// TwinCAT 3 PLC project VGR0
// ProgramVersion: 3.1.4024.0
// libraries:
//   Tc2_Standard, * (Beckhoff Automation GmbH)
//   Tc2_System, * (Beckhoff Automation GmbH)
//   Tc3_Module, * (Beckhoff Automation GmbH)
// project tree:
//   DUTs/ ST_Axis.TcDUT
//   GVLs/ Axis.TcGVL (not stored) (excluded from build), INPUT.TcGVL, OUTPUT.TcGVL, Settings.TcGVL, VGR.TcGVL
//   POUs/ AxisHorizontal.TcPOU, AxisRotate.TcPOU, AxisVertical.TcPOU, MAIN_10MS.TcPOU, MAIN_1MS.TcPOU, Motor_move.TcPOU, StateMachine.TcPOU
//   POUs/FBs/ AboutEqual.TcPOU, AxisMovementController.TcPOU, AxisReferencing.TcPOU, EncoderSignalProcessor.TcPOU, Motor_Direction.TcPOU, Motor_Enable.TcPOU
//   / VGR_10MS.TcTTO, VGR_1MS.TcTTO
// (motion and I/O tree: see PLC project vgr)
// real-time tasks:
//   TASK PlcTask: cycle T#10ms, priority 20, ADS port 350
//   TASK VGR_10MS: cycle T#10ms, priority 22, ADS port 352
//   TASK VGR_1MS: cycle T#1ms, priority 23, ADS port 353
// variable links:
//   VGR0/VGR0 Instance <-> Device 1 (EtherCAT)/Term 1 (EK1100)/Term 6 (EL5152)
//     VGR_10MS Inputs/INPUT.IW_VGR_CounterValueHorizontal <-> ENC Status compact Channel 2/Counter value
//     VGR_10MS Inputs/INPUT.IW_VGR_CounterValueVertical <-> ENC Status compact Channel 1/Counter value
//   VGR0/VGR0 Instance <-> Device 1 (EtherCAT)/Term 1 (EK1100)/Term 7 (EL5152)
//     VGR_10MS Inputs/INPUT.IW_VGR_CounterValueRotate <-> ENC Status compact Channel 1/Counter value

CONFIGURATION VGR0
    RESOURCE PLC ON TwinCAT3
        TASK VGR_10MS(INTERVAL := T#10ms, PRIORITY := 22);
        TASK VGR_1MS(INTERVAL := T#1ms, PRIORITY := 23);
        PROGRAM MAIN_10MS WITH VGR_10MS : MAIN_10MS;
        PROGRAM MAIN WITH VGR_10MS : MAIN;
        PROGRAM MAIN_1MS WITH VGR_1MS : MAIN_1MS;
    END_RESOURCE
END_CONFIGURATION

// ---- DUTs/ST_Axis.TcDUT
TYPE ST_Axis :
STRUCT
	uiCounterValue				  		: UINT;
	bSetCounter				 			: BOOL;
	uiSetCounterValue			 		: UINT := 0;
	iControl 							: INT; //VGR = PWM Motor M1 vertical axis enable at 10#32
	iPWM				 				: INT; //VGR = PWM Motor M1 vertical axis
	bJogMinus					 		: BOOL; //VGR - Q1 = Motor M1 vertical axis up
	bJogPlus					 		: BOOL; //VGR - Q2 = Motor M1 vertical axis down
END_STRUCT
END_TYPE

// ---- GVLs/INPUT.TcGVL
{attribute 'qualified_only'}
VAR_GLOBAL
IX_START AT %I*: BOOL;
IX_STOP AT %I*:	BOOL;
IW_VGR_CounterValueVertical  		AT %I* : UINT;
IW_VGR_CounterValueHorizontal  		AT %I* : UINT;
IW_VGR_CounterValueRotate  			AT %I* : UINT;

END_VAR

// ---- GVLs/OUTPUT.TcGVL
{attribute 'qualified_only'}
VAR_GLOBAL

QX_VGR_SetCounterVertical 			AT %Q* : BOOL;
QX_VGR_SetCounterHorizontal 		AT %Q* : BOOL;
QX_VGR_SetCounterRotate 			AT %Q* : BOOL;

QW_VGR_SetCounterValueVertical 		AT %Q* : UINT;
QW_VGR_SetCounterValueRotate 		AT %Q* : UINT;
QW_VGR_SetCounterValueHorizontal 	AT %Q* : UINT;

END_VAR

// ---- GVLs/Settings.TcGVL
{attribute 'qualified_only'}
VAR_GLOBAL
	bUseAxisVertical : BOOL := TRUE;
	bUseAxisHorizontal : BOOL := TRUE;
	bUseAxisRotate : BOOL := TRUE;
	
	CurrentState : STRING ;

	desiredSpeedVertical : INT := 5000;
	desiredSpeedHorizontal : INT := 5000;
	desiredSpeedRotation : INT := 5000;
	
	pickPositionVertical : UINT := 500;
	pickPositionHorizontal : UINT := 500;
	pickPositionRotation : UINT := 500;
	
	placePositionVertical : UINT := 100;
	placePositionHorizontal : UINT := 100;
	placePositionRotation : UINT := 200;
END_VAR

// ---- GVLs/VGR.TcGVL
{attribute 'qualified_only'}
VAR_GLOBAL

IX_VGR_RefSwitchVerticalAxis_I1 AT %I*: BOOL; //VGR - I1 = Reference switch vertical axis
IX_VGR_RefSwitchHorizontalAxis_I2 AT %I*: BOOL;//VGR - I2 = Reference switch horizontal axis
IX_VGR_RefSwitchRotate_I3 AT %I*: BOOL; //VGR - I3 = Reference switch rotate      

QX_VGR_M1_VerticalAxisUp_Q1 AT %Q* : BOOL; //VGR - Q1 = Motor M1 vertical axis up
QX_VGR_M1_VerticalAxisDown_Q2 AT %Q* : BOOL; //VGR - Q2 = Motor M1 vertical axis down
QX_VGR_M2_HorizontalAxisBackward_Q3 AT %Q* : BOOL; //VGR - Q3 = Motor M2 horizontal axis backward
QX_VGR_M2_HorizontalAxisForward_Q4 AT %Q* : BOOL; //VGR - Q4 = Motor M2 horizontal axis forward
QX_VGR_M3_RotateClockwise_Q5 AT %Q* : BOOL; //VGR - Q5 = Motor M3 rotate clockwise
QX_VGR_M3_RotateCounterclockwise_Q6 AT %Q* : BOOL; //VGR - Q6 = Motor M3 rotate counterclockwise
QX_VGR_Compressor_Q7 AT %Q* : BOOL; //VGR - Q7 = Compressor
QX_VGR_ValveVacuum_Q8 AT %Q* : BOOL; //VGR - Q8 = Valve vacuum
QW_VGR_PWM_Vertical_Control AT %Q* : INT; //VGR = PWM Motor M1 vertical axis enable
QW_VGR_PWM_Vertical_M1 AT %Q* : INT; //VGR = PWM Motor M1 vertical axis
QW_VGR_PWM_Horizontal_Control AT %Q* : INT; //VGR = PWM Motor M2 horizontal axis enable
QW_VGR_PWM_Horizontal_M2 AT %Q* : INT; //VGR = PWM Motor M2 horizontal axis
QW_VGR_PWM_Rotate_Control AT %Q* : INT; //VGR = PWM Motor M3 rotate axis enable
QW_VGR_PWM_Rotate_M3 AT %Q* : INT; //VGR = PWM Motor M3 rotate axis 	

(* UNUSED *)
IX_VGR_EncoderVerticalAxisImp1_B1 AT %I* : BOOL; //VGR - Vertical axis encoder - Channel A
IX_VGR_EncoderVerticalAxisImp2_B2 AT %I* : BOOL; //VGR - Vertical axis encoder - Channel B
IX_VGR_EncoderHorizontalAxisImp1_B3 AT %I* : BOOL; //VGR - Horizontal axis encoder - Channel A
IX_VGR_EncoderHorizontalAxisImp2_B4 AT %I* : BOOL; //VGR - Horizontal axis encoder - Channel B
IX_VGR_EncoderRotateImp1_B5 AT %I* : BOOL; //VGR - Rotational axis encoder - Channel A
IX_VGR_EncoderRotateImp2_B6 AT %I* : BOOL; //VGR - Rotational axis encoder - Channel B
END_VAR

// ---- POUs/MAIN_10MS.TcPOU
PROGRAM MAIN_10MS
VAR
	idle: BOOL;
	homing: BOOL;
	pick: BOOL;
	place: BOOL;
END_VAR

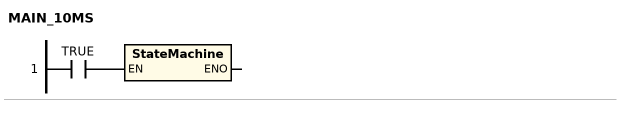
// NETWORK 1
StateMachine();

END_PROGRAM

// ---- POUs/StateMachine.TcPOU
PROGRAM StateMachine
VAR
	tolerance:UINT:=20;
	RS_Idle: RS;
	RS_Homing: RS;
	RS_place:RS;
	RS_Pick:RS;
	SR_ESTOP:SR;
	
	bValveClosed: BOOL;
	bValveOpen: BOOL;
	
	HorizontalState: AboutEqual;
	VerticalState: AboutEqual;
	RotationState: AboutEqual;
	bStateIdle: BOOL;
	bStateHoming: BOOL;
	bStatePick: BOOL;
	bStatePlace: BOOL;
	bStateEStop: BOOL;
	//check if position has reached
	Horizontal_Pick: BOOL;
	Vertical_Pick: BOOL;
	Rotation_Pick: BOOL;
	Horizontal_Place: BOOL;
	Vertical_Place: BOOL;
	Rotation_Place: BOOL;
	HorizontalState_b: AboutEqual;
	VerticalState_b: AboutEqual;
	RotationState_b: AboutEqual;
	HorizontalState_a: AboutEqual;
	VerticalState_a: AboutEqual;
	RotationState_a: AboutEqual;
END_VAR
VAR // added by the converter: edge detectors and wires of the graphical bodies
    _w1, _w2, _w3 : BOOL;
END_VAR

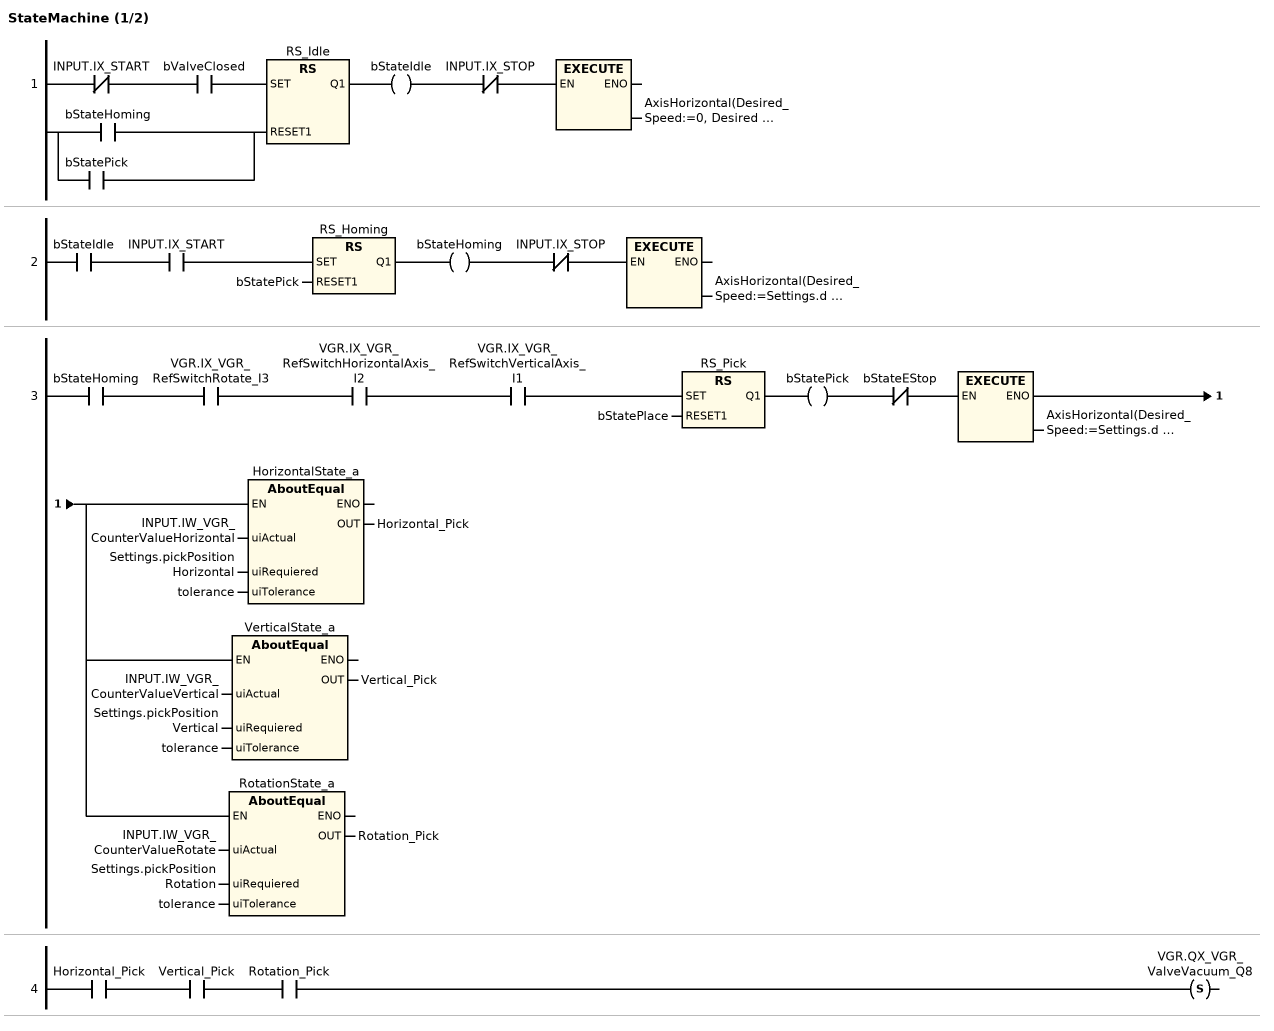
// NETWORK 1
RS_Idle(SET := NOT INPUT.IX_START AND bValveClosed, RESET1 := bStateHoming OR bStatePick); // RS
bStateIdle := RS_Idle.Q1;
IF RS_Idle.Q1 AND NOT INPUT.IX_STOP THEN
    AxisHorizontal(Desired_Speed:=0, Desired_Position:= input.IW_VGR_CounterValueHorizontal, tolerance:=20);
    AxisVertical(Desired_Speed:=0,
    			Desired_Position:= input.IW_VGR_CounterValueVertical,
    			tolerance:=20);
    AxisRotate(Desired_Speed:=0,
    			Desired_Position:= input.IW_VGR_CounterValueRotate,
    			tolerance:=20);
    Settings.CurrentState:='IDLE';
END_IF

// NETWORK 2
RS_Homing(SET := bStateIdle AND INPUT.IX_START, RESET1 := bStatePick); // RS
bStateHoming := RS_Homing.Q1;
IF RS_Homing.Q1 AND NOT INPUT.IX_STOP THEN
    AxisHorizontal(Desired_Speed:=Settings.desiredSpeedHorizontal,
    			Desired_Position:= 0,
    			tolerance:=tolerance);
    AxisVertical(Desired_Speed:=Settings.desiredSpeedVertical,
    			Desired_Position:= 0,
    			tolerance:=tolerance);
    AxisRotate(Desired_Speed:= Settings.desiredSpeedRotation,
    			Desired_Position:= 0,
    			tolerance:=tolerance);
    Settings.CurrentState:='HOME';
END_IF

// NETWORK 3
RS_Pick(SET := bStateHoming AND VGR.IX_VGR_RefSwitchRotate_I3 AND VGR.IX_VGR_RefSwitchHorizontalAxis_I2 AND VGR.IX_VGR_RefSwitchVerticalAxis_I1, RESET1 := bStatePlace); // RS
bStatePick := RS_Pick.Q1;
_w1 := RS_Pick.Q1 AND NOT bStateEStop;
IF _w1 THEN
    AxisHorizontal(Desired_Speed:=Settings.desiredSpeedHorizontal,
    			Desired_Position:= settings.pickPositionHorizontal,
    			tolerance:=tolerance);
    AxisVertical(Desired_Speed:=Settings.desiredSpeedVertical,
    			Desired_Position:= Settings.pickPositionVertical,
    			tolerance:=tolerance);
    AxisRotate(Desired_Speed:= Settings.desiredSpeedRotation,
    			Desired_Position:= settings.pickPositionRotation,
    			tolerance:=tolerance);
    Settings.CurrentState:='PICK';
END_IF
IF _w1 THEN
    HorizontalState_a(
        uiActual := INPUT.IW_VGR_CounterValueHorizontal,
        uiRequiered := Settings.pickPositionHorizontal,
        uiTolerance := tolerance,
        OUT => Horizontal_Pick); // AboutEqual
END_IF
IF _w1 THEN
    VerticalState_a(
        uiActual := INPUT.IW_VGR_CounterValueVertical,
        uiRequiered := Settings.pickPositionVertical,
        uiTolerance := tolerance,
        OUT => Vertical_Pick); // AboutEqual
END_IF
IF _w1 THEN
    RotationState_a(
        uiActual := INPUT.IW_VGR_CounterValueRotate,
        uiRequiered := Settings.pickPositionRotation,
        uiTolerance := tolerance,
        OUT => Rotation_Pick); // AboutEqual
END_IF

// NETWORK 4
VGR.QX_VGR_ValveVacuum_Q8 S= Horizontal_Pick AND Vertical_Pick AND Rotation_Pick;

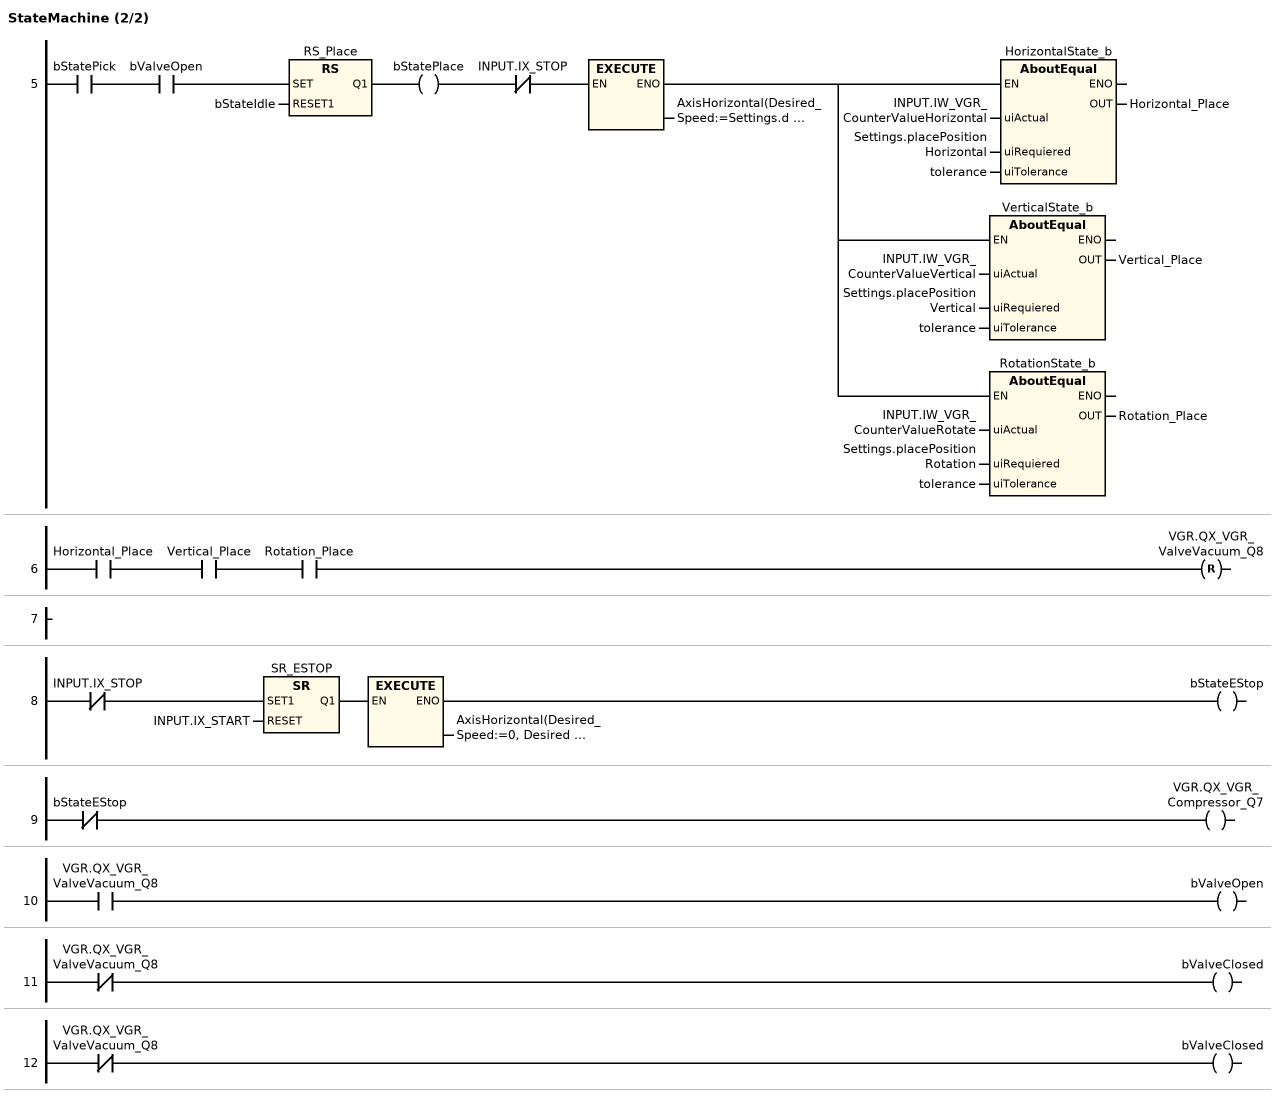
// NETWORK 5
RS_Place(SET := bStatePick AND bValveOpen, RESET1 := bStateIdle); // RS
bStatePlace := RS_Place.Q1;
_w2 := RS_Place.Q1 AND NOT INPUT.IX_STOP;
IF _w2 THEN
    AxisHorizontal(Desired_Speed:=Settings.desiredSpeedHorizontal,
    			Desired_Position:= Settings.placePositionHorizontal,
    			tolerance:=20);
    AxisVertical(Desired_Speed:=Settings.desiredSpeedVertical,
    			 Desired_Position:= Settings.placePositionVertical,
    	   		 tolerance:=20);
    AxisRotate(Desired_Speed:=Settings.desiredSpeedRotation,
    			Desired_Position:= Settings.placePositionRotation,
    			tolerance:=20);
    Settings.CurrentState:='PLACE';
END_IF
IF _w2 THEN
    HorizontalState_b(
        uiActual := INPUT.IW_VGR_CounterValueHorizontal,
        uiRequiered := Settings.placePositionHorizontal,
        uiTolerance := tolerance,
        OUT => Horizontal_Place); // AboutEqual
END_IF
IF _w2 THEN
    VerticalState_b(
        uiActual := INPUT.IW_VGR_CounterValueVertical,
        uiRequiered := Settings.placePositionVertical,
        uiTolerance := tolerance,
        OUT => Vertical_Place); // AboutEqual
END_IF
IF _w2 THEN
    RotationState_b(
        uiActual := INPUT.IW_VGR_CounterValueRotate,
        uiRequiered := Settings.placePositionRotation,
        uiTolerance := tolerance,
        OUT => Rotation_Place); // AboutEqual
END_IF

// NETWORK 6
VGR.QX_VGR_ValveVacuum_Q8 R= Horizontal_Place AND Vertical_Place AND Rotation_Place;

// NETWORK 7

// NETWORK 8
SR_ESTOP(SET1 := NOT INPUT.IX_STOP, RESET := INPUT.IX_START); // SR
_w3 := SR_ESTOP.Q1;
IF _w3 THEN
    AxisHorizontal(Desired_Speed:=0, Desired_Position:= input.IW_VGR_CounterValueHorizontal, tolerance:=20);
    AxisVertical(Desired_Speed:=0,
    			Desired_Position:= input.IW_VGR_CounterValueVertical,
    			tolerance:=20);
    AxisRotate(Desired_Speed:=0,
    			Desired_Position:= input.IW_VGR_CounterValueRotate,
    			tolerance:=20);
    Settings.CurrentState:='E_STOP';
END_IF
bStateEStop := _w3;

// NETWORK 9
VGR.QX_VGR_Compressor_Q7 := NOT bStateEStop;

// NETWORK 10
bValveOpen := VGR.QX_VGR_ValveVacuum_Q8;

// NETWORK 11
bValveClosed := NOT VGR.QX_VGR_ValveVacuum_Q8;

// NETWORK 12
bValveClosed := NOT VGR.QX_VGR_ValveVacuum_Q8;

END_PROGRAM

// ---- POUs/FBs/AboutEqual.TcPOU
FUNCTION_BLOCK AboutEqual
VAR_INPUT
	uiActual	: UINT;
	uiRequiered	: UINT;
	uiTolerance	: UINT;
END_VAR
VAR_OUTPUT
	OUT: BOOL;
END_VAR
VAR
	uiDifference: UINT;
END_VAR

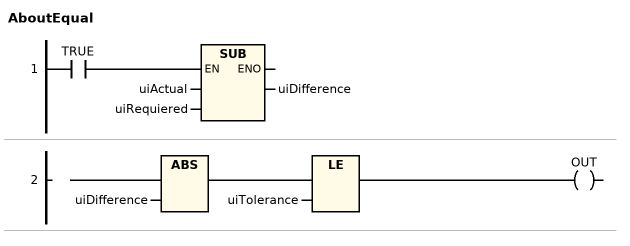
// NETWORK 1
uiDifference := uiActual - uiRequiered;

// NETWORK 2
OUT := ABS(uiDifference) <= uiTolerance;

END_FUNCTION_BLOCK

// ---- POUs/AxisHorizontal.TcPOU
PROGRAM AxisHorizontal
VAR_INPUT
	Desired_Speed: INT ;
	Desired_Position: UINT ;
	tolerance: UINT;
END_VAR
VAR
	Axis : ST_Axis := (
		uiCounterValue := INPUT.IW_VGR_CounterValueHorizontal,
		bSetCounter := OUTPUT.QX_VGR_SetCounterHorizontal,
		uiSetCounterValue := OUTPUT.QW_VGR_SetCounterValueHorizontal,
		iControl := VGR.QW_VGR_PWM_Horizontal_Control,
		iPWM := VGR.QW_VGR_PWM_Horizontal_M2,
		bJogMinus := VGR.QX_VGR_M2_HorizontalAxisBackward_Q3,
		bJogPlus := VGR.QX_VGR_M2_HorizontalAxisForward_Q4
	);
	Motor_Direction_Horizontal: Motor_direction;
END_VAR

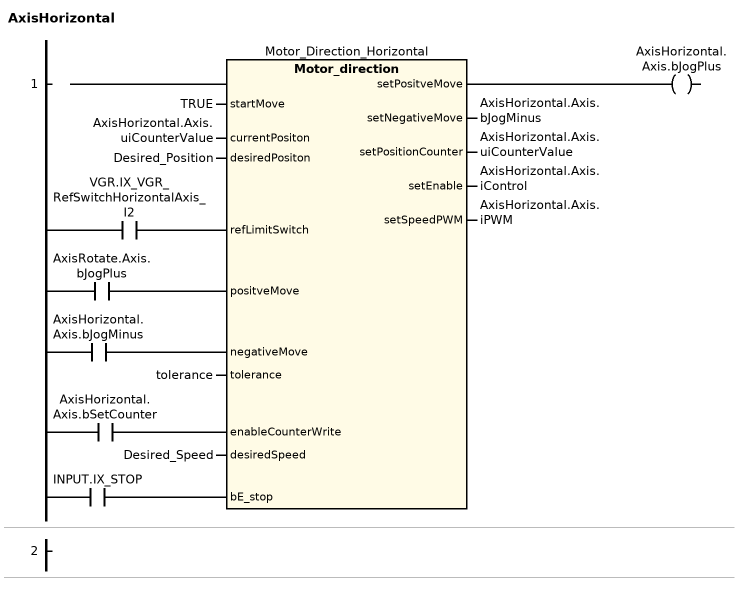
// NETWORK 1
Motor_Direction_Horizontal(
    startMove := TRUE,
    currentPositon := AxisHorizontal.Axis.uiCounterValue,
    desiredPositon := Desired_Position,
    refLimitSwitch := VGR.IX_VGR_RefSwitchHorizontalAxis_I2,
    positveMove := AxisRotate.Axis.bJogPlus,
    negativeMove := AxisHorizontal.Axis.bJogMinus,
    tolerance := tolerance,
    enableCounterWrite := AxisHorizontal.Axis.bSetCounter,
    desiredSpeed := Desired_Speed,
    bE_stop := INPUT.IX_STOP,
    setNegativeMove => AxisHorizontal.Axis.bJogMinus,
    setPositionCounter => AxisHorizontal.Axis.uiCounterValue,
    setEnable => AxisHorizontal.Axis.iControl,
    setSpeedPWM => AxisHorizontal.Axis.iPWM); // Motor_direction
AxisHorizontal.Axis.bJogPlus := Motor_Direction_Horizontal.setPositveMove;

// NETWORK 2

END_PROGRAM

// ---- POUs/FBs/Motor_Direction.TcPOU
FUNCTION_BLOCK Motor_Direction
VAR_INPUT
	startMove: BOOL;
	currentPositon: UINT;
	desiredPositon: UINT;
	refLimitSwitch: BOOL;
	positveMove: BOOL;
	negativeMove: BOOL;
	tolerance: UINT;
	enableCounterWrite: BOOL;
	desiredSpeed: INT;
	bE_stop: BOOL;
	//setEncoder: UINT;
	
END_VAR
VAR_OUTPUT
	setPositveMove: BOOL;
	setNegativeMove: BOOL;
	setPositionCounter: UINT;
	setEnable: INT;
	setSpeedPWM:INT;
END_VAR
VAR
	referencePosition: UINT :=0;
	
	motorEnable_vertival: Motor_Enable;
	
END_VAR

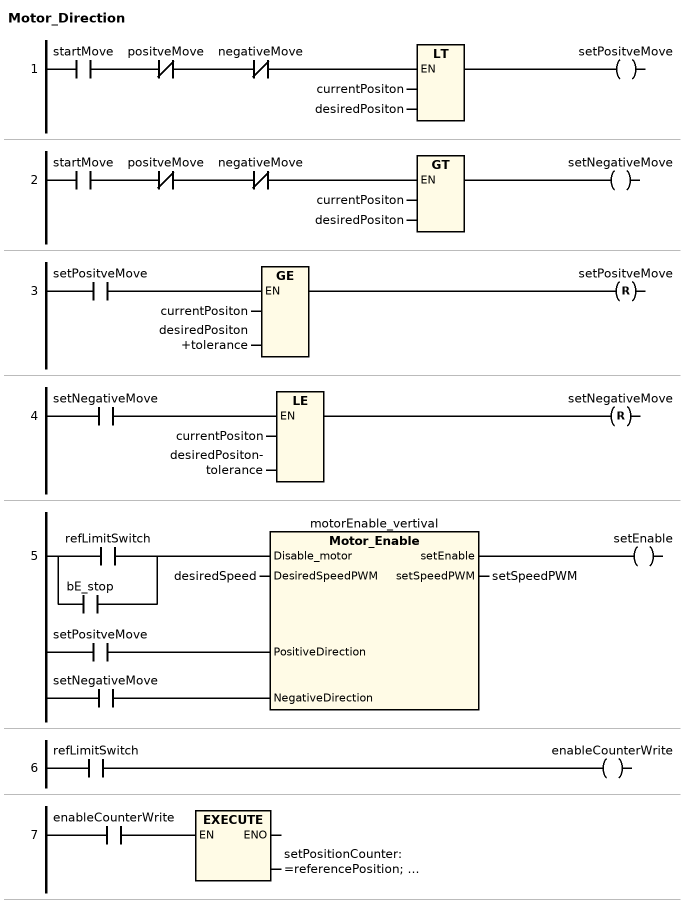
// NETWORK 1
setPositveMove := startMove AND NOT positveMove AND NOT negativeMove AND currentPositon < desiredPositon;

// NETWORK 2
setNegativeMove := startMove AND NOT positveMove AND NOT negativeMove AND currentPositon > desiredPositon;

// NETWORK 3
setPositveMove R= setPositveMove AND currentPositon >= (desiredPositon +tolerance);

// NETWORK 4
setNegativeMove R= setNegativeMove AND currentPositon <= (desiredPositon-tolerance);

// NETWORK 5
motorEnable_vertival(
    Disable_motor := refLimitSwitch OR bE_stop,
    DesiredSpeedPWM := desiredSpeed,
    PositiveDirection := setPositveMove,
    NegativeDirection := setNegativeMove,
    setSpeedPWM => setSpeedPWM); // Motor_Enable
setEnable := motorEnable_vertival.setEnable;

// NETWORK 6
enableCounterWrite := refLimitSwitch;

// NETWORK 7
IF enableCounterWrite THEN setPositionCounter:=referencePosition; END_IF

END_FUNCTION_BLOCK

// ---- POUs/FBs/Motor_Enable.TcPOU
FUNCTION_BLOCK Motor_Enable
VAR_INPUT
	Disable_motor: BOOL;
	DesiredSpeedPWM:INT;
	PositiveDirection: BOOL;
	NegativeDirection: BOOL;
END_VAR
VAR_OUTPUT
	setEnable: INT;
	setSpeedPWM:INT; 
END_VAR
VAR
	move_enabled: BOOL;
END_VAR
VAR // added by the converter: edge detectors and wires of the graphical bodies
    _w1, _w2 : BOOL;
END_VAR

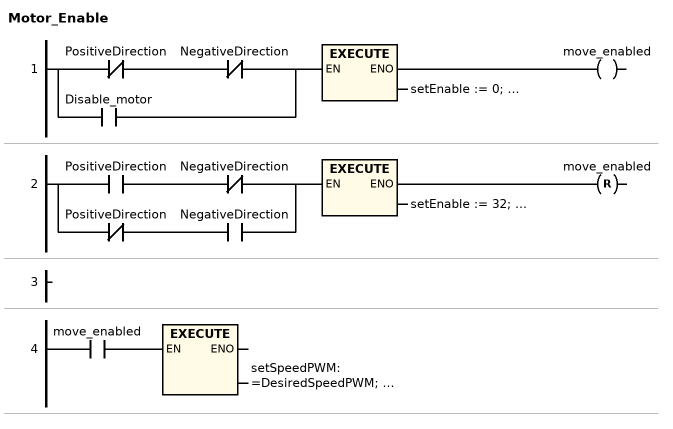
// NETWORK 1
_w1 := NOT PositiveDirection AND NOT NegativeDirection OR Disable_motor;
IF _w1 THEN
    setEnable := 0;
    setSpeedPWM:=0;
END_IF
move_enabled := _w1;

// NETWORK 2
_w2 := PositiveDirection AND NOT NegativeDirection OR NOT PositiveDirection AND NegativeDirection;
IF _w2 THEN setEnable := 32; END_IF
move_enabled R= _w2;

// NETWORK 3

// NETWORK 4
IF move_enabled THEN setSpeedPWM:=DesiredSpeedPWM; END_IF

END_FUNCTION_BLOCK

// ---- POUs/AxisRotate.TcPOU
PROGRAM AxisRotate
VAR_INPUT
	Desired_Speed: INT ;
	Desired_Position: UINT ;
	tolerance: UINT;
END_VAR
VAR
	Axis : ST_Axis := (
		uiCounterValue := INPUT.IW_VGR_CounterValueRotate,
		bSetCounter := OUTPUT.QX_VGR_SetCounterRotate,
		uiSetCounterValue := OUTPUT.QW_VGR_SetCounterValueRotate,
		iControl := VGR.QW_VGR_PWM_Rotate_Control,
		iPWM := VGR.QW_VGR_PWM_Rotate_M3,
		bJogMinus := VGR.QX_VGR_M3_RotateClockwise_Q5,
		bJogPlus := VGR.QX_VGR_M3_RotateCounterclockwise_Q6
	);
	Motor_Direction_Rotational: Motor_direction;
END_VAR

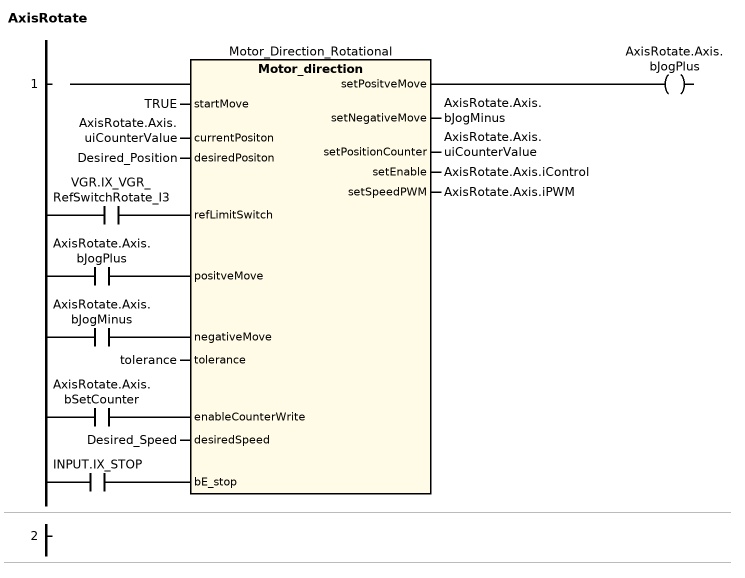
// NETWORK 1
Motor_Direction_Rotational(
    startMove := TRUE,
    currentPositon := AxisRotate.Axis.uiCounterValue,
    desiredPositon := Desired_Position,
    refLimitSwitch := VGR.IX_VGR_RefSwitchRotate_I3,
    positveMove := AxisRotate.Axis.bJogPlus,
    negativeMove := AxisRotate.Axis.bJogMinus,
    tolerance := tolerance,
    enableCounterWrite := AxisRotate.Axis.bSetCounter,
    desiredSpeed := Desired_Speed,
    bE_stop := INPUT.IX_STOP,
    setNegativeMove => AxisRotate.Axis.bJogMinus,
    setPositionCounter => AxisRotate.Axis.uiCounterValue,
    setEnable => AxisRotate.Axis.iControl,
    setSpeedPWM => AxisRotate.Axis.iPWM); // Motor_direction
AxisRotate.Axis.bJogPlus := Motor_Direction_Rotational.setPositveMove;

// NETWORK 2

END_PROGRAM

// ---- POUs/AxisVertical.TcPOU
PROGRAM AxisVertical
VAR_INPUT
	Desired_Speed: INT ;
	Desired_Position: UINT ;
	tolerance: UINT;
END_VAR
VAR
	Axis : ST_Axis := (
		uiCounterValue := INPUT.IW_VGR_CounterValueVertical,
		bSetCounter := OUTPUT.QX_VGR_SetCounterVertical,
		uiSetCounterValue := OUTPUT.QW_VGR_SetCounterValueVertical,
		iControl := VGR.QW_VGR_PWM_Vertical_Control,
		iPWM := VGR.QW_VGR_PWM_Vertical_M1,
		bJogMinus := VGR.QX_VGR_M1_VerticalAxisUp_Q1,
		bJogPlus := VGR.QX_VGR_M1_VerticalAxisDown_Q2
	);
	
	Motor_Direction_Vertical: Motor_direction;
END_VAR

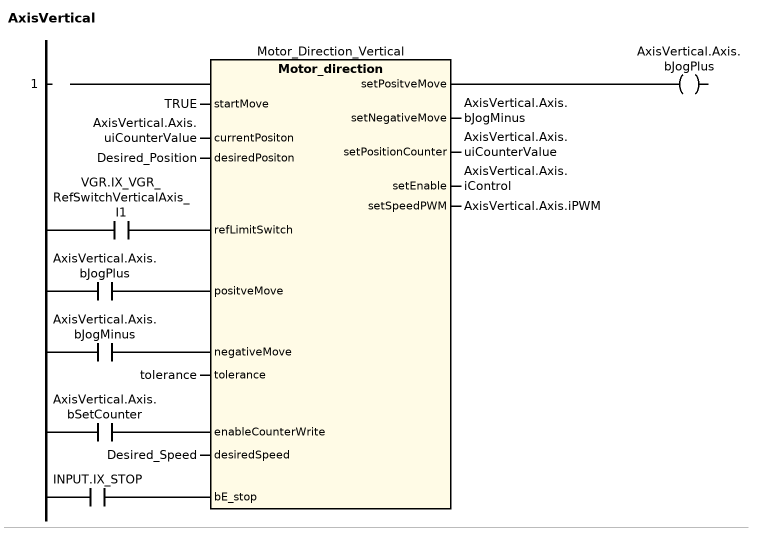
// NETWORK 1
Motor_Direction_Vertical(
    startMove := TRUE,
    currentPositon := AxisVertical.Axis.uiCounterValue,
    desiredPositon := Desired_Position,
    refLimitSwitch := VGR.IX_VGR_RefSwitchVerticalAxis_I1,
    positveMove := AxisVertical.Axis.bJogPlus,
    negativeMove := AxisVertical.Axis.bJogMinus,
    tolerance := tolerance,
    enableCounterWrite := AxisVertical.Axis.bSetCounter,
    desiredSpeed := Desired_Speed,
    bE_stop := INPUT.IX_STOP,
    setNegativeMove => AxisVertical.Axis.bJogMinus,
    setPositionCounter => AxisVertical.Axis.uiCounterValue,
    setEnable => AxisVertical.Axis.iControl,
    setSpeedPWM => AxisVertical.Axis.iPWM); // Motor_direction
AxisVertical.Axis.bJogPlus := Motor_Direction_Vertical.setPositveMove;

END_PROGRAM

// ---- POUs/MAIN_1MS.TcPOU
PROGRAM MAIN_1MS
VAR
END_VAR

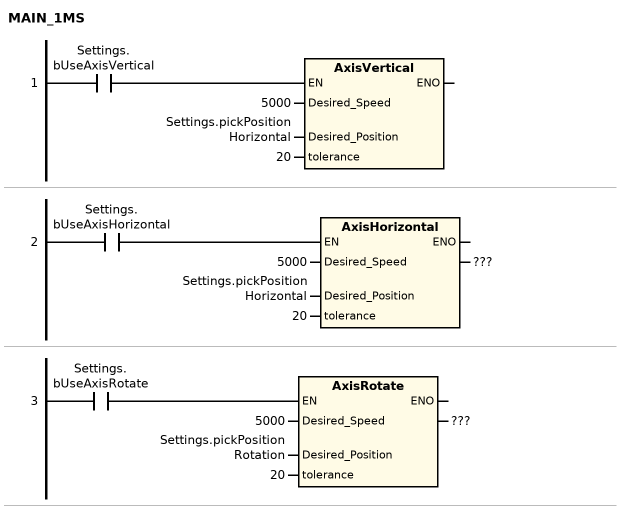
// NETWORK 1
IF Settings.bUseAxisVertical THEN
    AxisVertical(Desired_Speed := 5000, Desired_Position := Settings.pickPositionHorizontal, tolerance := 20);
END_IF

// NETWORK 2
IF Settings.bUseAxisHorizontal THEN
    AxisHorizontal(Desired_Speed := 5000, Desired_Position := Settings.pickPositionHorizontal, tolerance := 20);
END_IF

// NETWORK 3
IF Settings.bUseAxisRotate THEN
    AxisRotate(Desired_Speed := 5000, Desired_Position := Settings.pickPositionRotation, tolerance := 20);
END_IF

END_PROGRAM

// ---- POUs/FBs/AxisMovementController.TcPOU
FUNCTION_BLOCK AxisMovementController
VAR_INPUT
	tolerance: UINT;
	desiredSpeed: INT;
	currentPosition : UINT;
	requiredPosition : UINT;
END_VAR
VAR_OUTPUT
	AxisMinus : BOOL;
	AxisPlus: BOOL;
	Control: INT;
	SpeedPWM:INT;
	InPosition:BOOL;
END_VAR
VAR
END_VAR

IF  AboutEqual(
	uiActual:= currentPosition,
	uiRequiered:= requiredPosition,
	uiTolerance:= tolerance
)
 THEN
	AxisMinus := FALSE;
	AxisPlus := FALSE;
	Control := 0;
	SpeedPWM := 0;
	InPosition := TRUE;
ELSIF currentPosition > requiredPosition AND NOT InPosition THEN
	AxisMinus := TRUE;
	AxisPlus := FALSE;
	Control:= 32;
	SpeedPWM := desiredSpeed;
	InPosition := FALSE;
ELSIF currentPosition < requiredPosition AND NOT InPosition THEN
	AxisMinus := FALSE;
	AxisPlus := TRUE;
	Control := 32;
	SpeedPWM := desiredSpeed;
	InPosition := FALSE;
ELSE
	AxisMinus := FALSE;
	AxisPlus := FALSE;
	Control := 0;
	SpeedPWM := 0;
	InPosition := FALSE;
END_IF

END_FUNCTION_BLOCK

// ---- POUs/FBs/AxisReferencing.TcPOU
FUNCTION_BLOCK AxisReferencing
VAR_INPUT
	referencingSpeed: INT;
	ReferenceSwitch:BOOL;
END_VAR
VAR_OUTPUT
	AxisPlus:BOOL;
	AxisMinus:BOOL;
	Control:INT;
	SpeedPWM:INT;
	SetCounterValue: UINT;
	SetCounter:BOOL;
	ReferenceOkay:BOOL;
END_VAR
VAR
END_VAR

IF ReferenceSwitch THEN
	AxisMinus := FALSE;
	AxisPlus := FALSE;
	Control := 0;
	SpeedPWM := 0;
	SetCounter := TRUE;
	ReferenceOkay:= TRUE;
ELSE
	AxisMinus := TRUE;
	AxisPlus := FALSE;
	Control := 32;
	SetCounterValue := 0;
	SpeedPWM := referencingSpeed;
	SetCounter := FALSE;
END_IF

END_FUNCTION_BLOCK

// ---- POUs/FBs/EncoderSignalProcessor.TcPOU
FUNCTION_BLOCK EncoderSignalProcessor
VAR_INPUT
	pulseA : BOOL;
	pulseB : BOOL;
	//reset :	
	referencePositionSensor : BOOL;
	referencePosition: INT := 0;
END_VAR
VAR_OUTPUT
	direction : BOOL;
	position : INT;
END_VAR
VAR
	trigger : BOOL;
	direction_ : BOOL;
	count_ : INT;
	
END_VAR
VAR // added by the converter: edge detectors and wires of the graphical bodies
    _rt1, _rt2, _rt3, _rt4 : R_TRIG;
    _ft1, _ft2, _ft3, _ft4 : F_TRIG;
END_VAR

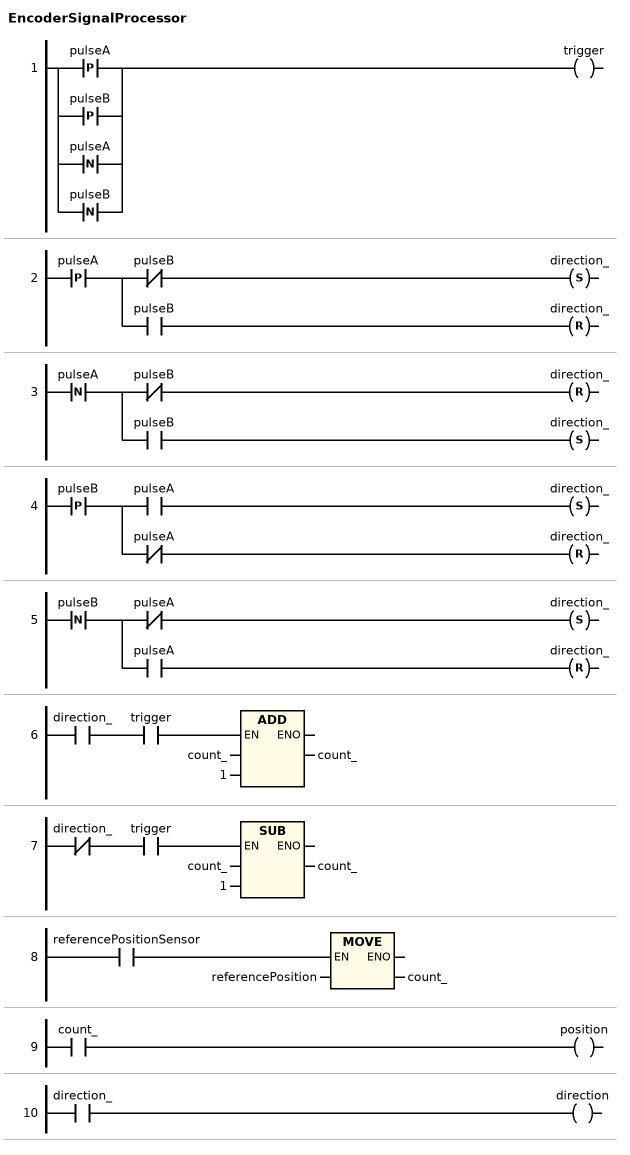
// NETWORK 1
_rt1(CLK := pulseA);
_rt2(CLK := pulseB);
_ft1(CLK := pulseA);
_ft2(CLK := pulseB);
trigger := _rt1.Q OR _rt2.Q OR _ft1.Q OR _ft2.Q;

// NETWORK 2
_rt3(CLK := pulseA);
direction_ S= _rt3.Q AND NOT pulseB;
direction_ R= _rt3.Q AND pulseB;

// NETWORK 3
_ft3(CLK := pulseA);
direction_ R= _ft3.Q AND NOT pulseB;
direction_ S= _ft3.Q AND pulseB;

// NETWORK 4
_rt4(CLK := pulseB);
direction_ S= _rt4.Q AND pulseA;
direction_ R= _rt4.Q AND NOT pulseA;

// NETWORK 5
_ft4(CLK := pulseB);
direction_ S= _ft4.Q AND NOT pulseA;
direction_ R= _ft4.Q AND pulseA;

// NETWORK 6
IF direction_ AND trigger THEN count_ := count_ + 1; END_IF

// NETWORK 7
IF NOT direction_ AND trigger THEN count_ := count_ - 1; END_IF

// NETWORK 8
IF referencePositionSensor THEN count_ := referencePosition; END_IF

// NETWORK 9
position := count_;

// NETWORK 10
direction := direction_;

END_FUNCTION_BLOCK

// ---- POUs/Motor_move.TcPOU
PROGRAM Motor_move
VAR
	motorDirection_rotate: Motor_Direction;
	position_rotation: UINT;
	writeRotateReference: BOOL;
	writeHorizontalReference: BOOL;
	writeVerticalReference: BOOL;
	tolerance: UINT :=20;
	movemotor_rotate: Motor_Enable;
	desiredSpeed: INT :=5000;
END_VAR

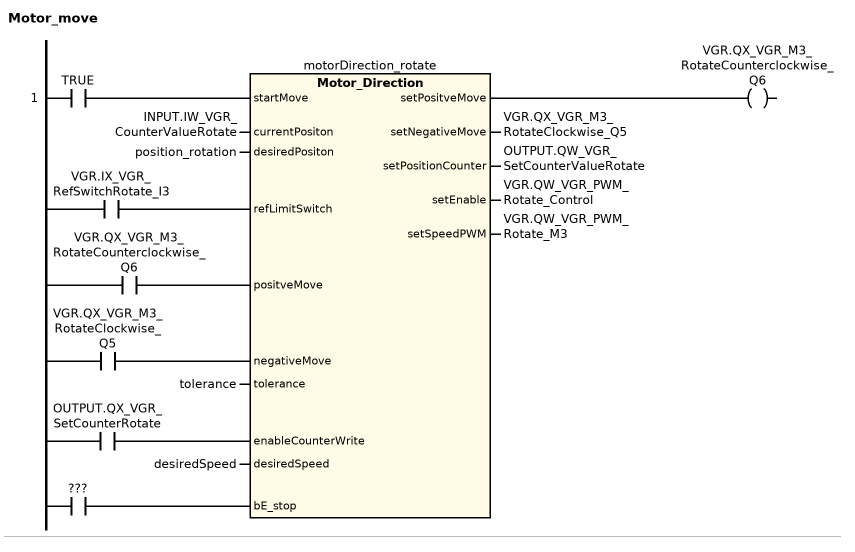
// NETWORK 1
motorDirection_rotate(
    startMove := TRUE,
    currentPositon := INPUT.IW_VGR_CounterValueRotate,
    desiredPositon := position_rotation,
    refLimitSwitch := VGR.IX_VGR_RefSwitchRotate_I3,
    positveMove := VGR.QX_VGR_M3_RotateCounterclockwise_Q6,
    negativeMove := VGR.QX_VGR_M3_RotateClockwise_Q5,
    tolerance := tolerance,
    enableCounterWrite := OUTPUT.QX_VGR_SetCounterRotate,
    desiredSpeed := desiredSpeed,
    setNegativeMove => VGR.QX_VGR_M3_RotateClockwise_Q5,
    setPositionCounter => OUTPUT.QW_VGR_SetCounterValueRotate,
    setEnable => VGR.QW_VGR_PWM_Rotate_Control,
    setSpeedPWM => VGR.QW_VGR_PWM_Rotate_M3); // Motor_Direction
VGR.QX_VGR_M3_RotateCounterclockwise_Q6 := motorDirection_rotate.setPositveMove;

END_PROGRAM
